// Slave Arm Base Controller, Hold at Current Posture
FUNCTION_BLOCK FB_SlaveArmCtrlBase IMPLEMENTS I_SlaveArmCtrl
VAR_INPUT
END_VAR
VAR_OUTPUT
END_VAR
VAR
	// flag if the controller has finished all its jobs
	m_isFinished:BOOL:=FALSE;
	
	// controller execute time period
	m_timePeriod :LREAL:=0;
	
	// flag to hold last commands
	m_holdLastCmds :BOOL := FALSE;
	
	// arm index
	m_armIdx: INT;
	
	// arm control data
	// NOTE: simulated joint position is usd for kinematic controller 
	//		while command joint position is used for real robot controller
	// 		They are identical for the most time, but in some cases, simulated position is filted to get command one 
	m_simJntPos :Vec8d; 
	m_cmdJntPos : VEC8d; 
	m_cmdJntVel : VEC8d;
	m_cmdJntAcc : VEC8d;
	m_cmdJntTrq : VEC8d;
	m_jntOPMode : Vec8i;
	m_jntEnableFlag :Vec8i;
	m_cmdCartPose : ST_Frame;
	m_cmdCartTwist : Vec6d;
	m_FFJntTrq :Vec8d;
	
END_VAR

// override this function in each exact controller
METHOD PROTECTED calcCmdJntPos : BOOL
VAR_IN_OUT CONSTANT
	// endoscope pose in cart coordinate
	i_endoscopePose : ST_Frame;
	
	// master arm data
	i_masterStatus :ST_MasterStatus;
	
	// setup arm data
	i_setupStatus: ST_SetupStatus;
	
	// slave arm data
	i_slaveArm :FB_SlaveArm;
END_VAR
IF isFinished THEN
	RETURN;
END_IF
END_METHOD

// override this function in each exact controller
METHOD PROTECTED calcCmdJntTrq : BOOL
VAR_IN_OUT CONSTANT
	// endoscope pose in cart coordinate
	i_endoscopePose : ST_Frame;
	
	// master arm data
	i_masterStatus :ST_MasterStatus;
	
	// setup arm data
	i_setupStatus: ST_SetupStatus;
	
	// slave arm data
	i_slaveArm :FB_SlaveArm;
END_VAR
IF isFinished THEN
	RETURN;
END_IF
END_METHOD

METHOD checkToHoldLastCmds : BOOL
VAR_IN_OUT CONSTANT
	i_slaveArm :FB_SlaveArm;
END_VAR
VAR
	j:INT;
	maxJntErr:LREAL;
	jntCtrlErr:Vec8d;
END_VAR
// check if to hold the command joint position unchanged
vecSub(i_slaveArm.m_cmdJntPos, i_slaveArm.m_curJntPos,jntCtrlErr);
maxJntErr:=0.0;
FOR j:=1 TO g_sJntNum DO
	maxJntErr:= MAX(maxJntErr, ABS(jntCtrlErr[j]));
END_FOR

checkToHoldLastCmds := (maxJntErr<GVL_SlaveControlParameters.g_jntCtrlErrForCmdHold);
END_METHOD

METHOD copyCmds : BOOL
VAR_IN_OUT 
	r_slaveArmCtrlCmd :ST_SlaveArmCtrlCmds;
END_VAR
r_slaveArmCtrlCmd.m_jntEnableFlag :=m_jntEnableFlag;
r_slaveArmCtrlCmd.m_cmdCartPose:=m_cmdCartPose;
r_slaveArmCtrlCmd.m_cmdCartTwist:=m_cmdCartTwist;
r_slaveArmCtrlCmd.m_simJntPos:=m_simJntPos;
r_slaveArmCtrlCmd.m_cmdJntPos:=m_cmdJntPos;
r_slaveArmCtrlCmd.m_cmdJntVel:=m_cmdJntVel;
r_slaveArmCtrlCmd.m_cmdJntAcc:=m_cmdJntAcc;
r_slaveArmCtrlCmd.m_cmdJntTrq:=m_cmdJntTrq;
r_slaveArmCtrlCmd.m_jntOPMode:=m_jntOPMode;
r_slaveArmCtrlCmd.m_FFJntTrq:=m_FFJntTrq;
END_METHOD

// call this function to add friction compensation to m_cmdJntTrq
METHOD enableFrictionCompensation : BOOL
VAR_IN_OUT CONSTANT
	i_slaveArm :FB_SlaveArm;
END_VAR

VAR
	i:INT;
	frictionScale :LREAL;
END_VAR
// add joint friction compensation
FOR i:=1 TO g_sJntNum DO
	frictionScale :=LIMIT(-1.0, i_slaveArm.curJntVel[i]/g_fullFrictionVel,1.0);
	m_cmdJntTrq[i]:=m_cmdJntTrq[i]+frictionScale * g_frictionCompScale * GVL_SlaveArmDynamics.g_slaveJntFriction[i_slaveArm.armIdx, i];
END_FOR
END_METHOD

// override this function in each exact controller
// NOTICE: set joint control mode here, and do some initialization if needed
METHOD PUBLIC init : BOOL
VAR_IN_OUT CONSTANT
	i_slaveArm	:FB_SlaveArm;
END_VAR
VAR_IN_OUT 
	r_slaveArmCtrlCmd :ST_SlaveArmCtrlCmds;
END_VAR
m_timePeriod:=0;
m_isFinished:=FALSE;
m_jntEnableFlag :=g_onesVec8i;
m_jntOPMode:=g_slaveAllPosTrqMode;
m_cmdCartPose:=i_slaveArm.curCartPose;
m_cmdCartTwist:=g_zeroVec6d;
IF FALSE = m_holdLastCmds THEN
	m_cmdJntPos:=i_slaveArm.curJntPos;
ELSE
	m_cmdJntPos:=r_slaveArmCtrlCmd.m_cmdJntPos;
END_IF
m_simJntPos := m_cmdJntPos;
m_cmdJntVel:=g_zeroVec8d;
m_cmdJntAcc:=g_zeroVec8d;
m_cmdJntTrq:=g_zeroVec8d;
m_FFJntTrq :=g_zeroVec8d;
m_armIdx:= i_slaveArm.armIdx;

// update commands to arm
copyCmds(r_slaveArmCtrlCmd);
END_METHOD

PROPERTY isFinished : BOOL
GET
isFinished:=m_isFinished;
END_GET
END_PROPERTY

{warning '添加方法实现'}
METHOD reset : BOOL
m_isFinished:=FALSE;
m_timePeriod:=0;
END_METHOD

{warning '添加方法实现'}
METHOD run : BOOL
VAR_IN_OUT CONSTANT
	i_endoscopePose : ST_Frame;
	i_masterStatus :ST_MasterStatus;
	i_setupStatus: ST_SetupStatus;
	i_slaveArm :FB_SlaveArm;
END_VAR
VAR_IN_OUT
	r_slaveArmCtrlCmd :ST_SlaveArmCtrlCmds;
END_VAR
VAR
	i:INT;
END_VAR
IF m_isFinished THEN
	RETURN;
END_IF

// check if arm enabled
IF FALSE = i_slaveArm.isEnabled(m_jntEnableFlag) THEN
	RETURN;
END_IF

// calculate command joint position--Motion control
calcCmdJntPos(i_endoscopePose, i_masterStatus, i_setupStatus, i_slaveArm);

// calculate command joint torque -- Force control
calcCmdJntTrq(i_endoscopePose, i_masterStatus, i_setupStatus, i_slaveArm);

// update commands to arm
copyCmds(r_slaveArmCtrlCmd);

// update time period
m_timePeriod := m_timePeriod+g_slaveArmCtrlCycleTime;
END_METHOD

PROPERTY timePeriod : Lreal
GET
timePeriod := m_timePeriod;
END_GET
END_PROPERTY

END_FUNCTION_BLOCK

(* stored: Version 1.1.0.1, ProductVersion 3.1.4024.12
   POU FB_SlaveArmCtrlBase: Id {dee0ec68-3abc-4720-b67c-0fb3fd57933b}, SpecialFunc None
   Folder Porperty: Id {c6953522-4b77-49b0-9e91-271eecbab135}
   Method calcCmdJntPos: Id {98ab3239-d030-4534-a55d-1eaac78d6af0}
   Method calcCmdJntTrq: Id {31ee0fe6-80c4-42e7-bd18-5b745e895642}
   Method checkToHoldLastCmds: Id {90f04ad1-6a41-4802-98b4-abd6341aeded}
   Method copyCmds: Id {5ed9a333-2aec-433d-86b7-210e62264fbb}
   Method enableFrictionCompensation: Id {10dd90f8-3406-4e7f-993e-818d061aef86}
   Method init: Id {63e02c69-11c3-4e06-9c58-dcaf1b3a881b}
   Property isFinished: Id {d6db4485-2c6d-406e-9b85-5a477e39dd21}
   Get Get: Id {438b47e5-c18c-4fc8-a8d2-2d2ca67eaf31}
   Method reset: Id {ac9e4b6b-f016-4e25-9efd-13892d3b6c48}
   Method run: Id {4a86d5bc-6efe-47db-8e4e-968f76a73eb3}
   Property timePeriod: Id {44038474-1ba7-4c9c-8c84-72a6505c50bc}
   Get Get: Id {a96f8ba3-aad3-45c7-b8fb-41d2e22f00f8} *)
